Omron CX-Programmer project NewProject (CX-Programmer 9.31)

# PLC NewPLC1: CP1L L

## Global symbols (name address type ; comment)
W0.06 BOOL  ; \
W0.07 BOOL  ; 13 hz
W0.08 BOOL  ; 15 hz
W0.09 BOOL  ; 10 hz

## Program NewProgram1 (cyclic task 0)

### Section Section1

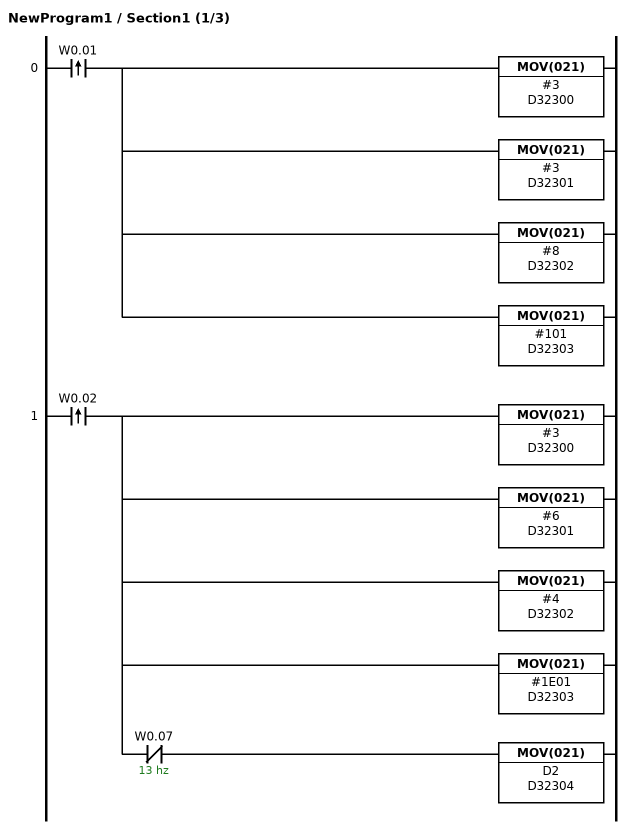
; rung 0
@LD W0.01
MOV(021) #3 D32300
MOV(021) #3 D32301
MOV(021) #8 D32302
MOV(021) #101 D32303
; rung 1
@LD W0.02
MOV(021) #3 D32300
MOV(021) #6 D32301
MOV(021) #4 D32302
MOV(021) #1E01 D32303
ANDNOT W0.07  ; 13 hz
MOV(021) D2 D32304

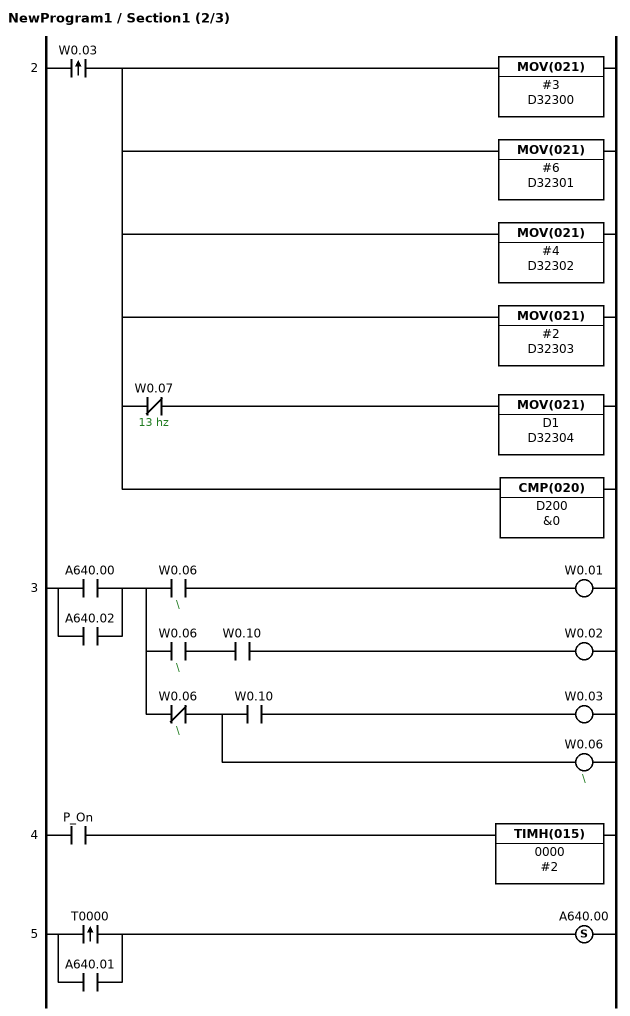
; rung 2
@LD W0.03
OUT TR0
MOV(021) #3 D32300
MOV(021) #6 D32301
MOV(021) #4 D32302
MOV(021) #2 D32303
ANDNOT W0.07  ; 13 hz
MOV(021) D1 D32304
LD TR0
CMP(020) D200 &0
; rung 3
LD A640.00
OR A640.02
OUT TR0
AND W0.06  ; \
OUT W0.01
LD TR0
AND W0.06  ; \
AND W0.10
OUT W0.02
LD TR0
ANDNOT W0.06  ; \
OUT TR0
AND W0.10
OUT W0.03
LD TR0
OUT W0.06  ; \
; rung 4
LD P_On
TIMH(015) 0000 #2
; rung 5
@LD T0000
OR A640.01
SET A640.00

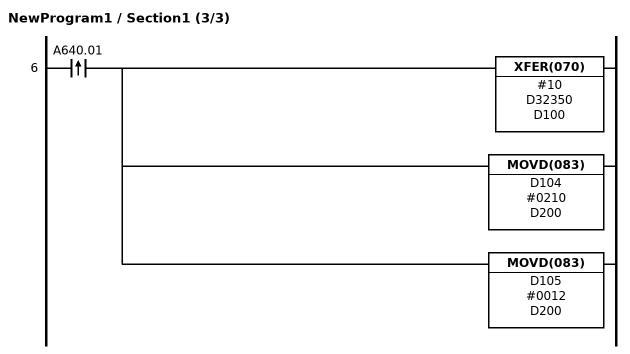
; rung 6
@LD A640.01
XFER(070) #10 D32350 D100
MOVD(083) D104 #0210 D200
MOVD(083) D105 #0012 D200

### Section END
; rung 0
END(001)